// TIA Portal V17 export
// export: Created 2025-06-26T06:49:34.3187458Z, ExportSetting WithDefaults, DisplayName Totally Integrated Automation Portal, DisplayVersion V17 Update 8, DisplayName TIA Portal Openness, DisplayVersion V17 Update 8, DisplayName TIA Portal Version Control Interface, DisplayVersion V17, DisplayName STEP 7 Professional, DisplayVersion V17 Update 8, DisplayName STEP 7 Safety, DisplayVersion V17 Update 6, DisplayName WinCC Advanced, DisplayVersion V17 Update 8
VAR_GLOBAL   // PLC tag table "RIO2"
   RIO2_Slot4_I AT %I934.0 : "stSM531_8AI";   //    {ExternalAccessible false, ExternalVisible false, ExternalWritable false}
   RIO2_Slot2_I AT %I900.0 : "stSM531_8AI";   //    {ExternalAccessible false, ExternalVisible false, ExternalWritable false}
   RIO2_Slot3_I AT %I917.0 : "stSM531_8AI";   //    {ExternalAccessible false, ExternalVisible false, ExternalWritable false}
   RIO2_Slot5_I AT %I951.0 : "stSM531_8AI";   //    {ExternalAccessible false, ExternalVisible false, ExternalWritable false}
   RIO2_Slot6_I AT %I968.0 : "stSM531_8AI";   //    {ExternalAccessible false, ExternalVisible false, ExternalWritable false}
   RIO2_Slot7_I AT %I985.0 : "stSM531_8AI";   //    {ExternalAccessible false, ExternalVisible false, ExternalWritable false}
   RIO2_Slot8_I AT %I1002.0 : "stSM531_8AI";   //    {ExternalAccessible false, ExternalVisible false, ExternalWritable false}
   RIO2_Slot9_I AT %I1019.0 : "stSM531_8AI";   //    {ExternalAccessible false, ExternalVisible false, ExternalWritable false}
   RIO2_Slot10_I AT %I1036.0 : "stSM531_8AI";   //    {ExternalAccessible false, ExternalVisible false, ExternalWritable false}
   RIO2_Slot11_I AT %I1053.0 : "stSM531_8AI";   //    {ExternalAccessible false, ExternalVisible false, ExternalWritable false}
   RIO2_Slot12_I AT %I1070.0 : "stSM531_8AI";   //    {ExternalAccessible false, ExternalVisible false, ExternalWritable false}
   RIO2_Slot13_I AT %I1087.0 : "stSM521_16DI";   //    {ExternalAccessible false, ExternalVisible false, ExternalWritable false}
   RIO2_Slot14_I AT %I1089.0 : "stSM531_8AQ_I";   //    {ExternalAccessible false, ExternalVisible false, ExternalWritable false}
   RIO2_Slot15_I AT %I1090.0 : "stSM531_8AQ_I";   //    {ExternalAccessible false, ExternalVisible false, ExternalWritable false}
   RIO2_Slot16_I AT %I1091.0 : "stSM522_32DQ_I";   //    {ExternalAccessible false, ExternalVisible false, ExternalWritable false}
   RIO2_Slot14_Q AT %Q900.0 : "stSM531_8AQ";   //    {ExternalAccessible false, ExternalVisible false, ExternalWritable false}
   RIO2_Slot15_Q AT %Q916.0 : "stSM531_8AQ";   //    {ExternalAccessible false, ExternalVisible false, ExternalWritable false}
   RIO2_Slot16_Q AT %Q932.0 : "stSM522_32DQ_Q";   //    {ExternalAccessible false, ExternalVisible false, ExternalWritable false}
END_VAR
